// SIMATIC S7-200 SMART project (STEP 7-Micro/WIN SMART), CPU SR40

SYMBOL_TABLE Table 1
SEALMANCMD       M0.0
PULLFILMMANCMD   M0.1
PRODOUTMANCMD    M0.2
AUTORUN          M0.3
SensorIn         M0.4
NormalCycle      M0.5
ProdInStart      M0.6
ProdInStop       M0.7
ProdOutStart     M1.0
ProdOutStop      M1.1
InitProdInStart  M1.2
InitProdOutStart M1.3
SealingStart     M1.4
SealingDone      M1.5
SealAutoCmd      M1.6
SealLimitError   M1.7
UnwindCmd        M2.0
ProdPassed       M2.1
OutConvStart     M2.2
END_SYMBOL_TABLE

ORGANIZATION_BLOCK MAIN:OB1
TITLE=Program Comments
BEGIN
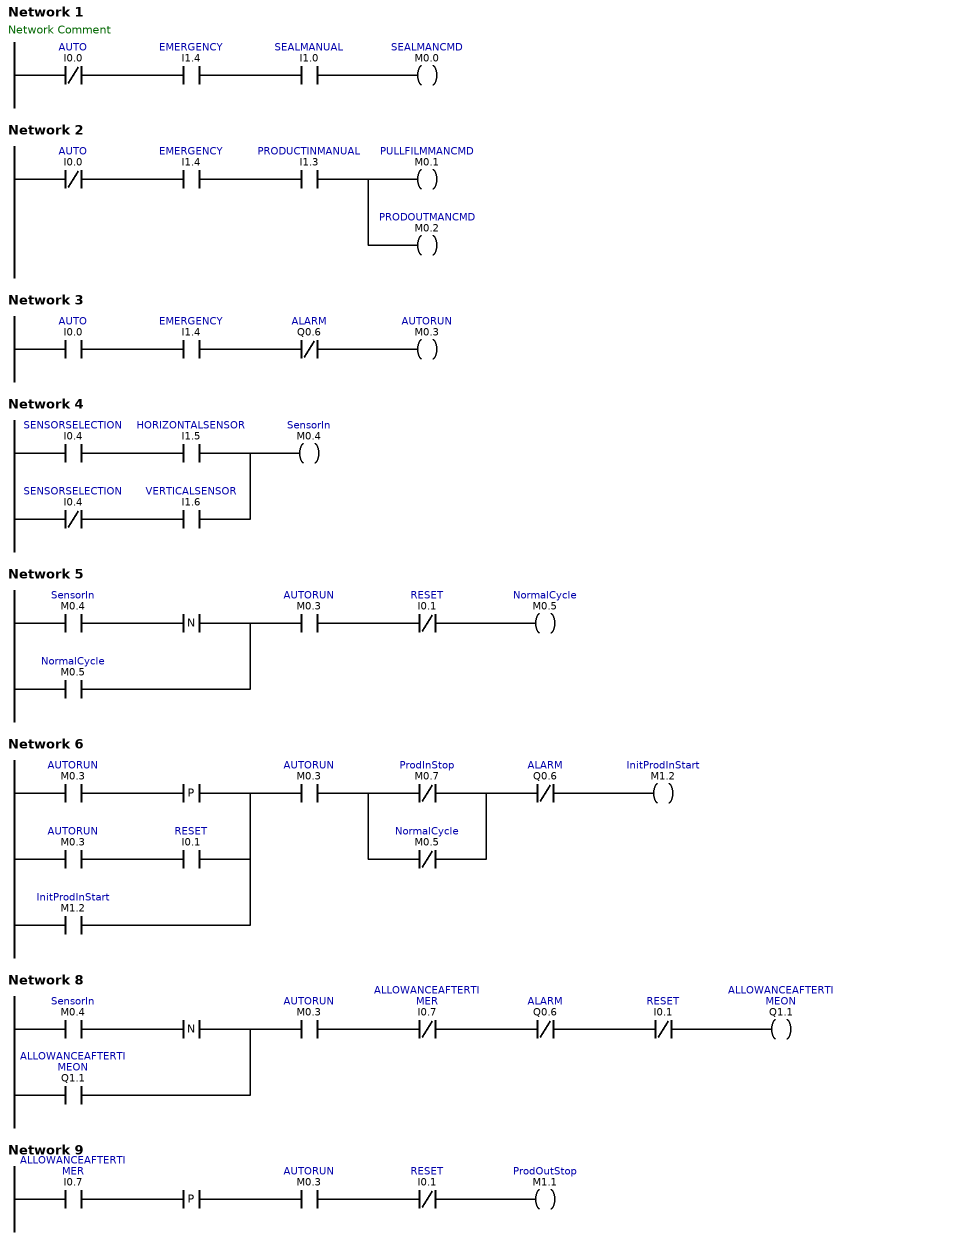
Network 1
// Network Comment
LDN    AUTO:I0.0
A      EMERGENCY:I1.4
A      SEALMANUAL:I1.0
=      SEALMANCMD:M0.0
Network 2
LDN    AUTO:I0.0
A      EMERGENCY:I1.4
A      PRODUCTINMANUAL:I1.3
=      PULLFILMMANCMD:M0.1
=      PRODOUTMANCMD:M0.2
Network 3
LD     AUTO:I0.0
A      EMERGENCY:I1.4
AN     ALARM:Q0.6
=      AUTORUN:M0.3
Network 4
LD     SENSORSELECTION:I0.4
A      HORIZONTALSENSOR:I1.5
LDN    SENSORSELECTION:I0.4
A      VERTICALSENSOR:I1.6
OLD
=      SensorIn:M0.4
Network 5
LD     SensorIn:M0.4
ED
O      NormalCycle:M0.5
A      AUTORUN:M0.3
AN     RESET:I0.1
=      NormalCycle:M0.5
Network 6
LD     AUTORUN:M0.3
EU
LD     AUTORUN:M0.3
A      RESET:I0.1
OLD
O      InitProdInStart:M1.2
A      AUTORUN:M0.3
LDN    ProdInStop:M0.7
ON     NormalCycle:M0.5
ALD
AN     ALARM:Q0.6
=      InitProdInStart:M1.2
Network 8
LD     SensorIn:M0.4
ED
O      ALLOWANCEAFTERTIMEON:Q1.1
A      AUTORUN:M0.3
AN     ALLOWANCEAFTERTIMER:I0.7
AN     ALARM:Q0.6
AN     RESET:I0.1
=      ALLOWANCEAFTERTIMEON:Q1.1
Network 9
LD     ALLOWANCEAFTERTIMER:I0.7
EU
A      AUTORUN:M0.3
AN     RESET:I0.1
=      ProdOutStop:M1.1
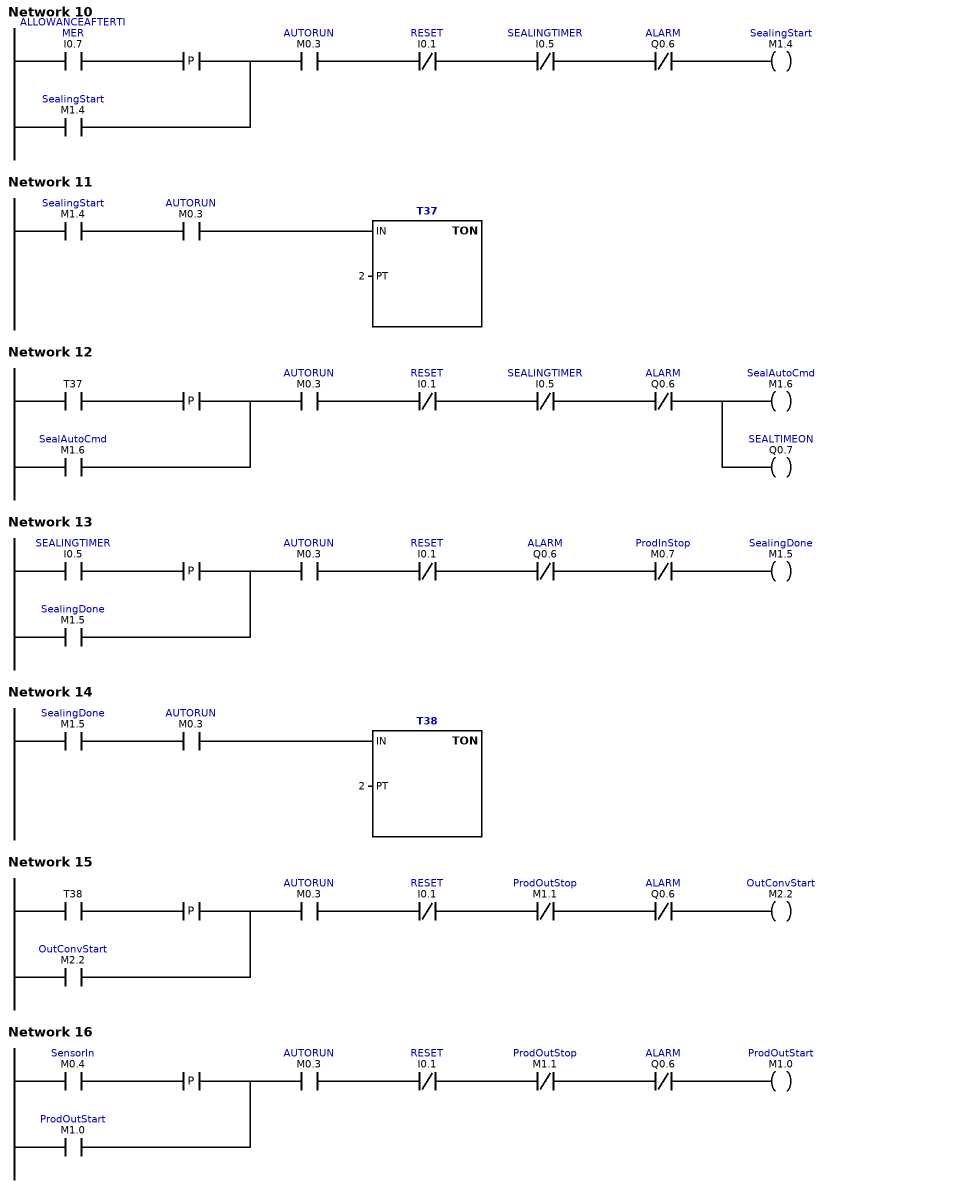
Network 10
LD     ALLOWANCEAFTERTIMER:I0.7
EU
O      SealingStart:M1.4
A      AUTORUN:M0.3
AN     RESET:I0.1
AN     SEALINGTIMER:I0.5
AN     ALARM:Q0.6
=      SealingStart:M1.4
Network 11
LD     SealingStart:M1.4
A      AUTORUN:M0.3
TON    T37, 2
Network 12
LD     T37
EU
O      SealAutoCmd:M1.6
A      AUTORUN:M0.3
AN     RESET:I0.1
AN     SEALINGTIMER:I0.5
AN     ALARM:Q0.6
=      SealAutoCmd:M1.6
=      SEALTIMEON:Q0.7
Network 13
LD     SEALINGTIMER:I0.5
EU
O      SealingDone:M1.5
A      AUTORUN:M0.3
AN     RESET:I0.1
AN     ALARM:Q0.6
AN     ProdInStop:M0.7
=      SealingDone:M1.5
Network 14
LD     SealingDone:M1.5
A      AUTORUN:M0.3
TON    T38, 2
Network 15
LD     T38
EU
O      OutConvStart:M2.2
A      AUTORUN:M0.3
AN     RESET:I0.1
AN     ProdOutStop:M1.1
AN     ALARM:Q0.6
=      OutConvStart:M2.2
Network 16
LD     SensorIn:M0.4
EU
O      ProdOutStart:M1.0
A      AUTORUN:M0.3
AN     RESET:I0.1
AN     ProdOutStop:M1.1
AN     ALARM:Q0.6
=      ProdOutStart:M1.0
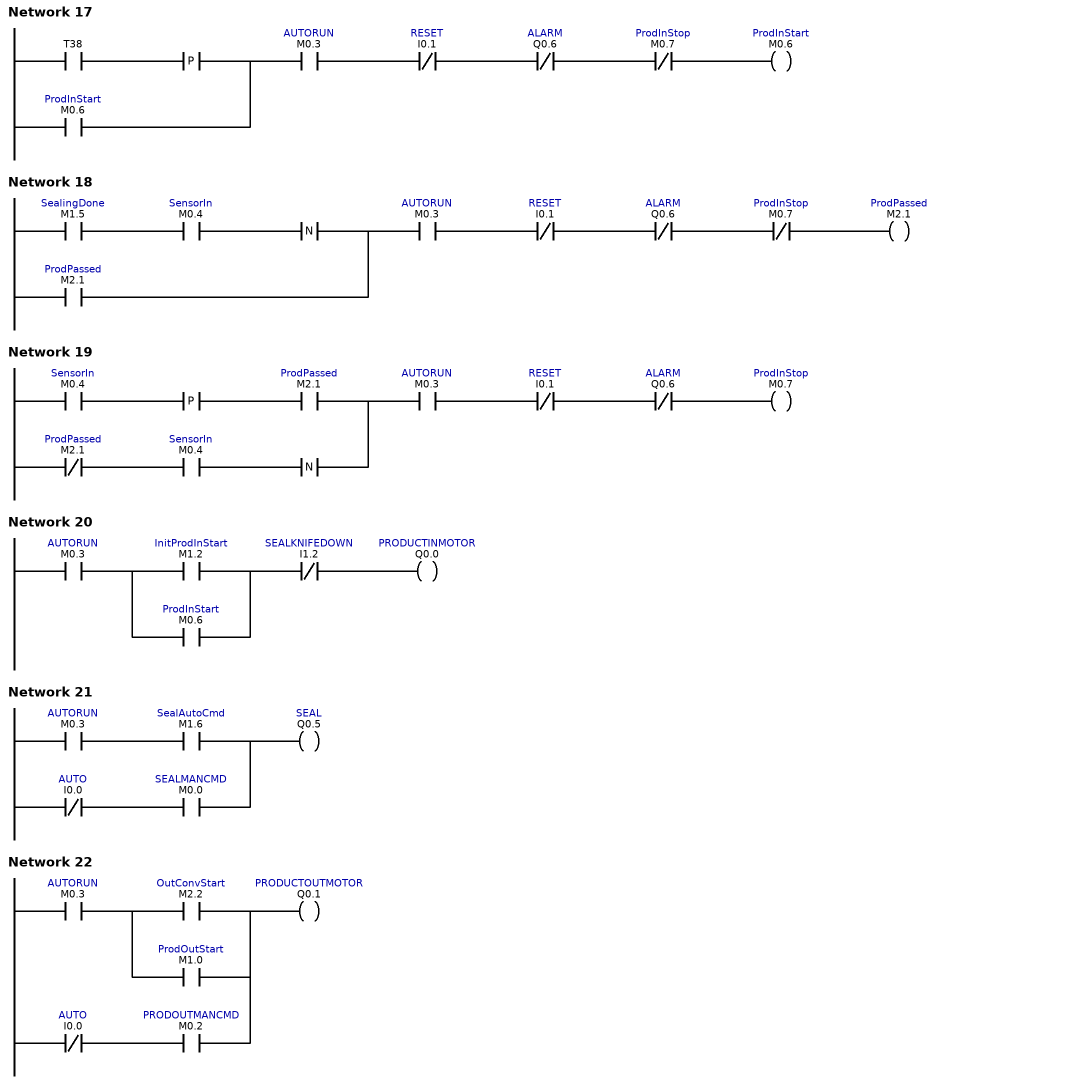
Network 17
LD     T38
EU
O      ProdInStart:M0.6
A      AUTORUN:M0.3
AN     RESET:I0.1
AN     ALARM:Q0.6
AN     ProdInStop:M0.7
=      ProdInStart:M0.6
Network 18
LD     SealingDone:M1.5
A      SensorIn:M0.4
ED
O      ProdPassed:M2.1
A      AUTORUN:M0.3
AN     RESET:I0.1
AN     ALARM:Q0.6
AN     ProdInStop:M0.7
=      ProdPassed:M2.1
Network 19
LD     SensorIn:M0.4
EU
A      ProdPassed:M2.1
LDN    ProdPassed:M2.1
A      SensorIn:M0.4
ED
OLD
A      AUTORUN:M0.3
AN     RESET:I0.1
AN     ALARM:Q0.6
=      ProdInStop:M0.7
Network 20
LD     AUTORUN:M0.3
LD     InitProdInStart:M1.2
O      ProdInStart:M0.6
ALD
AN     SEALKNIFEDOWN:I1.2
=      PRODUCTINMOTOR:Q0.0
Network 21
LD     AUTORUN:M0.3
A      SealAutoCmd:M1.6
LDN    AUTO:I0.0
A      SEALMANCMD:M0.0
OLD
=      SEAL:Q0.5
Network 22
LD     AUTORUN:M0.3
LD     OutConvStart:M2.2
O      ProdOutStart:M1.0
ALD
LDN    AUTO:I0.0
A      PRODOUTMANCMD:M0.2
OLD
=      PRODUCTOUTMOTOR:Q0.1
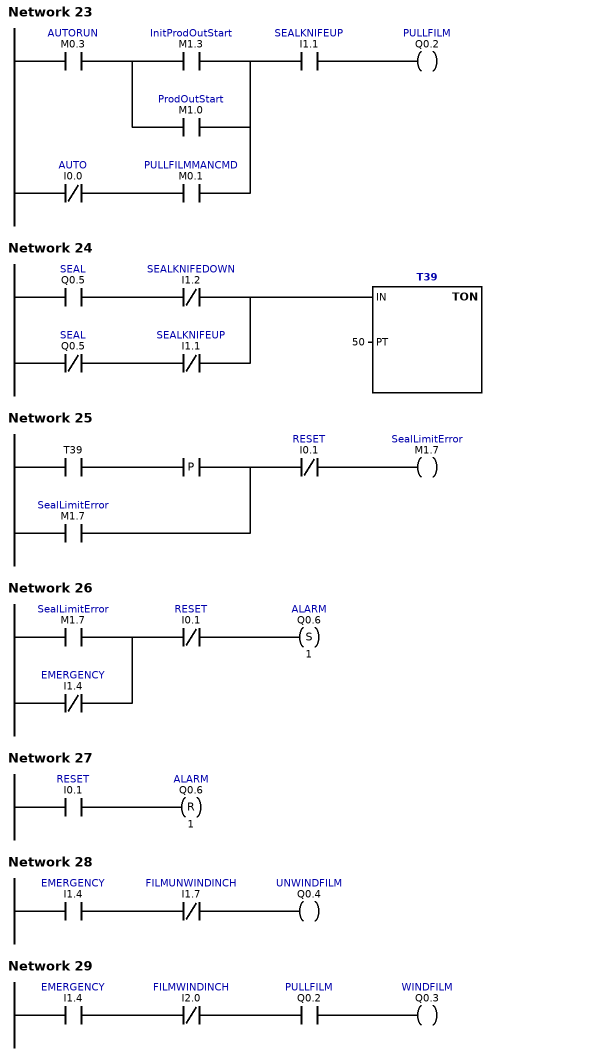
Network 23
LD     AUTORUN:M0.3
LD     InitProdOutStart:M1.3
O      ProdOutStart:M1.0
ALD
LDN    AUTO:I0.0
A      PULLFILMMANCMD:M0.1
OLD
A      SEALKNIFEUP:I1.1
=      PULLFILM:Q0.2
Network 24
LD     SEAL:Q0.5
AN     SEALKNIFEDOWN:I1.2
LDN    SEAL:Q0.5
AN     SEALKNIFEUP:I1.1
OLD
TON    T39, 50
Network 25
LD     T39
EU
O      SealLimitError:M1.7
AN     RESET:I0.1
=      SealLimitError:M1.7
Network 26
LD     SealLimitError:M1.7
ON     EMERGENCY:I1.4
AN     RESET:I0.1
S      ALARM:Q0.6, 1
Network 27
LD     RESET:I0.1
R      ALARM:Q0.6, 1
Network 28
LD     EMERGENCY:I1.4
AN     FILMUNWINDINCH:I1.7
=      UNWINDFILM:Q0.4
Network 29
LD     EMERGENCY:I1.4
AN     FILMWINDINCH:I2.0
A      PULLFILM:Q0.2
=      WINDFILM:Q0.3
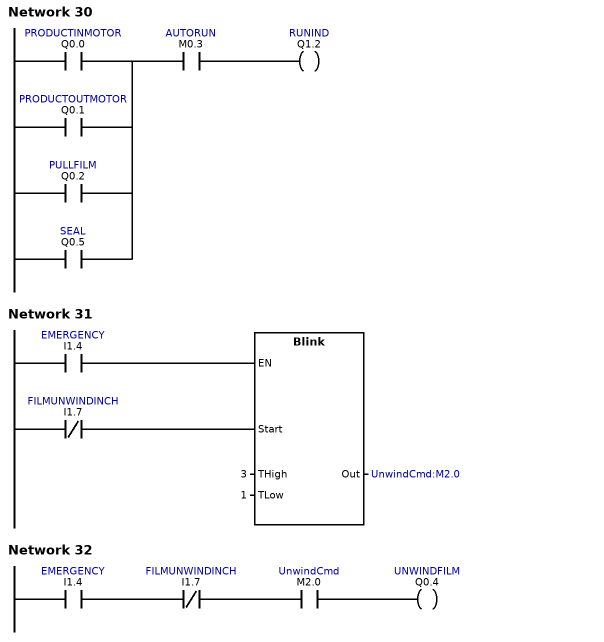
Network 30
LD     PRODUCTINMOTOR:Q0.0
O      PRODUCTOUTMOTOR:Q0.1
O      PULLFILM:Q0.2
O      SEAL:Q0.5
A      AUTORUN:M0.3
=      RUNIND:Q1.2
Network 31
LD     EMERGENCY:I1.4
=      L60.0
LDN    FILMUNWINDINCH:I1.7
=      L63.7
LD     L60.0
CALL   Blink:SBR1, L63.7, 3, 1, UnwindCmd:M2.0
Network 32
LD     EMERGENCY:I1.4
AN     FILMUNWINDINCH:I1.7
A      UnwindCmd:M2.0
=      UNWINDFILM:Q0.4
END_ORGANIZATION_BLOCK

// SBR1: protected block, not included
